(* CODESYS project wago_curl_post_example_v0.0.1.ecp

Project tree, tasks and I/O mapping:
  PFC100_2ETH_1 : 750-8101 PFC100 CS 2ETH, WAGO, order no. 0750-8101, version 5.11.1.16
    application Application
      libraries: ; SysProcess, 3.5.7.0 (System); ISysTypes2, 3.5.0.0 (System); WagoAppFileDir, * (WAGO)
      task PLC_Task (cyclic, interval t#50ms, priority 15) calls PLC_PRG
      function block fb_cURL_post_insecure [ST]: meth_cURL_post
      program PLC_PRG [ST]
      function fun_values_to_JSON [ST]
    DeviceAdapter
    Kbus : Kbus, WAGO, version 1.4.0.2
        unmapped channels: K-BUS diagnostics
      _2AO_4_20mA_1 : 0750-0554, WAGO, order no. 0750-0554, version 0.0.0.9
          settings: K-BUS Module slot index = 1
          unmapped channels: _QW 1, _QW 2
        DeviceAdapter
      _8AI_0_4_20mA_SE_1 : 0750-0496, WAGO, order no. 0750-0496, version 0.0.0.9
          settings: K-BUS Module slot index = 2
          unmapped channels: _PW 1, _PW 2, _PW 3, _PW 4, _PW 5, _PW 6, _PW 7, _PW 8
        DeviceAdapter
    MODBUS
      MODBUS : MODBUS, WAGO, order no. n/a, version 1.1.1.15
    Serial
*)

// PFC100_2ETH_1/Application/PLC_PRG
PROGRAM PLC_PRG
VAR
	sCurlData	: STRING(255); 
	iId			: INT := 10;
	iValue		: INT := 123;
	sTimeStamp	: STRING := '2018-01-01 01:01:09';
	fbCurlPost	: fb_cURL_post_insecure;
	xCurlPost: BOOL;
END_VAR

sCurlData := fun_values_to_JSON(INT_TO_STRING(iId), INT_TO_STRING(iValue), sTimeStamp);

fbCurlPost(
	sDataString:= sCurlData, 
	sEndPoint:= '<yourEndpoint>', 
	xExecute:= xCurlPost);

END_PROGRAM

// PFC100_2ETH_1/Application/fun_values_to_JSON
FUNCTION fun_values_to_JSON : STRING(255)
VAR_INPUT
	// {"auxDataPointTypeId":10, "value":3, "effectiveDate":"2017-10-01 02:99:99”} 
	sAuxDataPointTypeId		: STRING(80);
	sValue					: STRING(80);
	sEffectiveDate			: STRING(80);
END_VAR
VAR
	sHoldString				: STRING(255);
END_VAR

sHoldString := '{"auxDataPointTypeId" : ';						//{"auxDataPointTypeId" : 
sHoldString := CONCAT(sHoldString, sAuxDataPointTypeId);		//{"auxDataPointTypeId":10
sHoldString := CONCAT(sHoldString, ', "value" : ');				//{"auxDataPointTypeId":10, "value":
sHoldString := CONCAT(sHoldString, sValue);						//{"auxDataPointTypeId":10, "value":3
sHoldString := CONCAT(sHoldString, ', "effectiveDate" : "');	//{"auxDataPointTypeId":10, "value":3, "effectiveDate":"
sHoldString := CONCAT(sHoldString, sEffectiveDate);				//{"auxDataPointTypeId":10, "value":3, "effectiveDate":"2017-10-01 02:99:99
sHoldString := CONCAT(sHoldString, '"}');						//{"auxDataPointTypeId":10, "value":3, "effectiveDate":"2017-10-01 02:99:99”}

fun_values_to_JSON := sHoldString;								// writes the hold string to the output of the function

END_FUNCTION

// PFC100_2ETH_1/Application/fb_cURL_post_insecure
FUNCTION_BLOCK fb_cURL_post_insecure
VAR_INPUT
	sDataString	: STRING(255);	// this is the data to send
	sEndPoint	: STRING(255);	// the URL to send the data
END_VAR
VAR_IN_OUT
	xExecute	: BOOL;	// execute toggles off when fb is complete
END_VAR
VAR_OUTPUT
	// no output as of yet - could add some timeouts for the file system
END_VAR
VAR
	fbWriteFile	: WagoAppFileDir.FbWriteWholeFile_cpt;
	oWriteFileStatus: FbResult;
	xWriteFileTrigger: BOOL;
	xWriteFileError: BOOL;
	xWriteFileBusy: BOOL;
	sWriteStatus: STRING(255);
	diFileStatus: DINT;
	sCurlString: STRING(255);
END_VAR

IF xExecute THEN
	IF NOT xWriteFileTrigger THEN
		xWriteFileTrigger := TRUE;
	END_IF
	fbWriteFile(
		oStatus=> oWriteFileStatus, 
		xTrigger:= xWriteFileTrigger, 
		xError=> xWriteFileError, 
		xBusy=> xWriteFileBusy, 
		sName:= '/root/curldata.json', 
		pTxBuffer:= ADR(sDataString), 
		udiTxNBytes:= LEN(sDataString));
		
		IF NOT xWriteFileBusy AND NOT xWriteFileTrigger THEN
			xWriteFileTrigger := FALSE;
			sWriteStatus := meth_cURL_post('/root/curldata.json', sEndPoint);
			xExecute := FALSE;
		END_IF
END_IF

METHOD meth_cURL_post : STRING(255)
VAR_INPUT
	sFilePath	: STRING(255);
	sEndPoint	: STRING(255);
END_VAR
VAR 
	sCurlString	: STRING(255);// := 'curl --insecure --output /root/weather.json -X GET http://api.wunderground.com/api/';	// base string to query weather service
	pRslt: POINTER TO RTS_IEC_RESULT;
	ptBashRslt: POINTER TO RTS_IEC_RESULT;
END_VAR
sCurlString := 'curl -X POST --insecure -T ';
sCurlString := CONCAT(sCurlString, sFilePath);
sCurlString := CONCAT(sCurlString, ' ');
sCurlString := CONCAT(sCurlString, sEndpoint);

diFileStatus := SysProcessExecuteCommand(sCurlString, ptBashRslt);
END_METHOD

END_FUNCTION_BLOCK
